	fbExtensionTimeout_TON(IN := bExtending, PT := tExtensionTimeout);	//Timer for monitoring extension timeout, PT = Extension time multiplied by the timeout factor
	fbRetractionTimeout_TON(IN := bRetracting, PT := tRetractionTimeout);	//Timer for monitoring retraction timeout, PT = Retraction time multiplied by the timeout factor

	//Simultaneous extend and retract commands throw an invalid command error
	IF 		(bExtending AND bRetracting)
		OR 	(bExtendRequest AND bRetractRequest)
		OR 	(bExtendCommand AND bRetractCommand) THEN 
		nErrorID := E_CylinderBase.InvalidCommand;
	END_IF
	
	//If both extended and retracted feedback are true at any point, throw an invalid position error
	IF bExtended AND bRetracted THEN
		bError := TRUE;
		nErrorID := E_CylinderBase.InvalidPositionStatus;
	END_IF
	
	//If the cylinder takes longer than expected to extend, throw a timeout error
	IF fbExtensionTimeout_TON.Q THEN
		bError := TRUE;
		nErrorID := E_CylinderBase.ExtendTimeout;
	END_IF
	
	//If the cylinder takes longer than expected to retract, throw a timeout error
	IF fbRetractionTimeout_TON.Q THEN
		bError := TRUE;
		nErrorID := E_CylinderBase.RetractTimeout;
	END_IF
END_IF

//If cylinder is in motion toward a position, but it has not yet been reached, set busy bit
IF (bExtending) OR (bRetracting) THEN
	bActive := TRUE;
ELSE
	bActive := FALSE;
END_IF

IF bSimExtendCommand OR bExtendCommand THEN
	bExtendOutput := TRUE;
ELSE
	bExtendOutput := FALSE;
END_IF

IF bSimRetractCommand OR bRetractCommand THEN
	bRetractOutput := TRUE;
ELSE
	bRetractOutput := FALSE;
END_IF
END_METHOD

METHOD Reset : BOOL
SUPER^.Reset();

bExtending := FALSE;
bRetracting := FALSE;

fbSimExtend_TON.IN := FALSE;
fbSimRetract_TON.IN := FALSE;

bExtendCommand := FALSE;
bRetractCommand := FALSE;
END_METHOD

METHOD Retract : UDINT
bRetractRequest := TRUE;
bExtendRequest := FALSE;
bIncomingRequest := TRUE;
END_METHOD

PROPERTY Retracted : BOOL	//Status bit for the position of the cylinder
GET
Retracted := bRetracted;
END_GET
END_PROPERTY

PROPERTY Retracting : BOOL
GET
Retracting := bRetracting;
END_GET
END_PROPERTY

PROPERTY RetractOutput : BOOL
GET
RetractOutput := bRetractOutput;
END_GET
END_PROPERTY

PROPERTY RetractTime : TIME
GET
RetractTime := tRetractTime;
END_GET
SET
tRetractTime := RetractTime;
END_SET
END_PROPERTY

METHOD SimulateOperation : BOOL
VAR_INPUT
END_VAR
IF bEnabled THEN
	
	bExtendCommand := FALSE;		//Hardware commands should be disabled during simulation mode
	bRetractCommand := FALSE;		//Hardware commands should be disabled during simulation mode
	
	fbSimExtend_TON();		//Call timer FB
	fbSimRetract_TON();		//Call timer FB
	
	IF fbSimExtend_TON.Q THEN		//Whenever the extend timer completes, set status to extended and turn off the timer
		bExtended := TRUE;
		fbSimExtend_TON.IN := FALSE;
	END_IF
	
	IF fbSimRetract_TON.Q THEN		//Whenever the retract timer completes, set status to retracted and turn off the timer
		bRetracted := TRUE;
		fbSimRetract_TON.IN := FALSE;
	END_IF
	
	IF bIncomingRequest THEN
		IF bExtendRequest THEN					//Whenever a new extend request comes in, check to see if we are still currently timing a retract action
			IF fbSimRetract_TON.IN THEN			//If a retract action is still in progress, appropriately scale the extend time to account for the distance traveled during the in-process retraction
				fbSimExtend_TON.PT := tExtendTime * (TIME_TO_UDINT(fbSimRetract_TON.ET) / TIME_TO_UDINT(tRetractTime));		//partial extend time = (full distance extend time) * (proportional distance covered during retraction)
				bSimRetractCommand := FALSE;
				fbSimRetract_TON.IN := FALSE;	//Disable retract timer
			ELSE
				fbSimExtend_TON.PT := tExtendTime;	//If no retraction was active, assume we are currently at fully retracted position, or this is the first command the cylinder has received, so initialize to full extend time
			END_IF
			bRetracted := FALSE;
			bSimRetractCommand := FALSE;
			bSimExtendCommand := TRUE;
			fbSimExtend_TON.IN := TRUE;				//Activate the extension timer
		ELSIF bRetractRequest THEN					//Same as above, but reversed
			IF fbSimExtend_TON.IN THEN
				fbSimRetract_TON.PT := tRetractTime * (TIME_TO_UDINT(fbSimExtend_TON.ET) / TIME_TO_UDINT(tRetractTime));
				bSimExtendCommand := FALSE;
				fbSimExtend_TON.IN := FALSE;
			ELSE
				fbSimRetract_TON.PT := tRetractTime;
			END_IF
			bExtended := FALSE;
			fbSimRetract_TON.IN := TRUE;
			bSimExtendCommand := FALSE;
			bSimRetractCommand := TRUE;
		ELSE
			bExtended := FALSE;
			bRetracted := FALSE;
			
			fbSimExtend_TON.IN := FALSE;			
			fbSimRetract_TON.IN := FALSE;
			
			bSimExtendCommand := FALSE;
			bSimRetractCommand := FALSE;
		END_IF
		bIncomingRequest := FALSE;
	END_IF
	
	bExtending := fbSimExtend_TON.IN;
	bRetracting := fbSimRetract_TON.IN;
ELSE
	bIncomingRequest := FALSE;
	fbSimExtend_TON.IN := FALSE;
	fbSimRetract_TON.IN := FALSE;
END_IF
END_METHOD

METHOD StandardOperation : BOOL
VAR_INPUT
END_VAR
IF bEnabled THEN
	IF bIncomingRequest THEN
		bExtendCommand := bExtendRequest;
		bRetractCommand := bRetractRequest;
		bIncomingRequest := FALSE;
	END_IF
	
	IF bExtendCommand AND NOT bExtended THEN
		bExtending := TRUE;
	END_IF
	
	IF bRetractCommand AND NOT bRetracted THEN
		bRetracting := TRUE;
	END_IF
	
	bExtended := bExtendedFeedback;
	bRetracted := bRetractedFeedback;
ELSE
	bIncomingRequest := FALSE;
END_IF
END_METHOD

PROPERTY TimeoutFactor : LREAL	//Multiplicative factor that determines error timeout threshold based on the expected time
GET
TimeoutFactor := fTimeoutFactor;
END_GET
SET
fTimeoutFactor := TimeoutFactor;
END_SET
END_PROPERTY

END_FUNCTION_BLOCK

// ---- Base/02_Components/01_Base/FB_ComponentBase.TcPOU
FUNCTION_BLOCK FB_ComponentBase IMPLEMENTS ITF_ComponentBase
VAR_INPUT
END_VAR
VAR_OUTPUT
END_VAR
VAR CONSTANT
	//Constant declarations
	COMPONENT_BASE_ALARM_COUNT	: UDINT := 16;
END_VAR

VAR	
	//ITF_BasicComponent internal property variables
	bError 			: BOOL;			//Boolean to signal that an error has ocurred
	nErrorID 		: UDINT;		//Integer ID to identify the proper alarm to be posted from the parent module
	bEnabled		: BOOL;			//Enables or disables the component
	bSimulate		: BOOL;			//TRUE disables all hardware I/O and simulates input and output behavior
	sName			: STRING;		//String name of the component
	bActive			: BOOL;			//TRUE when the component is in its energized state, motion or detection
	
	//Alarming
	a_fbComponentBaseAlarms : ARRAY[1..COMPONENT_BASE_ALARM_COUNT] OF FB_TcAlarm;
	
	//HMI Monitoring and control structure
	stComponentBaseHMI : ST_ComponentBase_HMI;
	
	//Internal Variables
	bInitialized	: BOOL;
	
END_VAR

PROPERTY Active : BOOL	//TRUE when the component is in motion or otherwise completing a commanded task
GET
Active := bActive;
END_GET
END_PROPERTY

METHOD CyclicLogic : BOOL		//Should be called Externally akin to the PML Modules
IF NOT bInitialized THEN
	initialize();
	bInitialized := TRUE;
END_IF

IF NOT bSimulate AND NOT bError THEN	//If not in simulation mode or error state
	StandardOperation();
ELSIF NOT bError THEN
	SimulateOperation();	//Simulate inputs and outputs
ELSE
	ErrorOperation();
END_IF

Monitoring();		//Constant error and status monitoring
HardwareUpdate();	//Passes internal commands to hardware outputs and vice versa for inputs, implement via extended FB override
HMICommunication();	//Keeps the HMI data up to date, and processes requests from the HMI for this component
END_METHOD

PROPERTY Enabled : BOOL	//Enables or disables the component
GET
Enabled := bEnabled;
END_GET
SET
bEnabled := Enabled;
END_SET
END_PROPERTY

PROPERTY Error : BOOL	//Boolean to signal that an error has ocurred
GET
Error := bError;
END_GET
END_PROPERTY

PROPERTY ErrorID : UDINT	//Integer ID to identify the proper alarm to be posted from the parent module
GET
ErrorID := nErrorID;
END_GET
SET
nErrorID := ErrorID;
END_SET
END_PROPERTY

METHOD ErrorOperation : BOOL
VAR_INPUT
END_VAR
//Override from extended FB with error operation logic (Shut off outputs, clear inputs, blink, send error messages, etc)
END_METHOD

METHOD HardwareUpdate : BOOL
VAR_INPUT
END_VAR
//override from extended FB with reads and writes between internal variables and hardware inputs and outputs
END_METHOD

METHOD HMICommunication : BOOL
//Extend this method in extended FBs to communicate specific implementation data

//Process HMI requests
IF stComponentBaseHMI.bIncomingHMIRequest AND NOT stComponentBaseHMI.bHMICommandConfirmation THEN		//If a request has been issued by the HMI, and a previous request has not just finished being processed
	IF stComponentBaseHMI.bHMIControlAvailable THEN		//If the current conditions permit HMI control (Should be determined by the extended application components)
		IF stComponentBaseHMI.bEnableHMIRequest THEN
			bEnabled := TRUE;
			stComponentBaseHMI.bHMICommandConfirmation := TRUE;	//Confirm that the request has been processed
		END_IF
		IF stComponentBaseHMI.bDisableHMIRequest THEN
			bEnabled := FALSE;
			stComponentBaseHMI.bHMICommandConfirmation := TRUE;	//Confirm that the request has been processed
		END_IF
		IF stComponentBaseHMI.bResetHMIRequest THEN
			Reset();
			stComponentBaseHMI.bHMICommandConfirmation := TRUE;	//Confirm that the request has been processed
		END_IF
		IF stComponentBaseHMI.bSimulateOperationHMIRequest THEN
			bSimulate := TRUE;
			stComponentBaseHMI.bHMICommandConfirmation := TRUE;	//Confirm that the request has been processed
		END_IF
		IF stComponentBaseHMI.bStandardOperationHMIRequest THEN
			bSimulate := FALSE;
			stComponentBaseHMI.bHMICommandConfirmation := TRUE;	//Confirm that the request has been processed
		END_IF
	END_IF
END_IF

//Update HMI status info
stComponentBaseHMI.bActive := bActive;
stComponentBaseHMI.bEnabled := bEnabled;
stComponentBaseHMI.sName := sName;
stComponentBaseHMI.bError := bError;
stComponentBaseHMI.bSimulate := bSimulate;
stComponentBaseHMI.nErrorID := nErrorID;
END_METHOD

METHOD initialize : BOOL
VAR_INPUT
END_VAR

VAR
	sTemp: STRING;
END_VAR
//Extend initialize as needed in extended FBs

sTemp := CONCAT(CONCAT(CONCAT('Component ', ': '), sName), ' '); 	//Creates a utility string for alarms and other messaging that reads (example text) - "Module 10 - Main Casepacker" to be followed by the alarm or message info
//TODO: Rename Event Class to AxisBase
F_CreateAllEventsInClass(	p_aAlarms := a_fbComponentBaseAlarms,
							nClassSize := SIZEOF(TC_EVENTS.ComponentBase),
							pInitEvent := ADR(TC_EVENTS.ComponentBase.InitReferenceEvent),
							sPrefix := sTemp );
END_METHOD

METHOD Monitoring : BOOL
VAR_INPUT
END_VAR
//Override/extend from extended FB with monitoring logic
END_METHOD

PROPERTY Name : STRING
GET
Name := sName;
END_GET
SET
sName := Name;
END_SET
END_PROPERTY

METHOD Reset : BOOL
bError := FALSE;
nErrorID := 0;
END_METHOD

{warning 'add property implementation'}
PROPERTY Simulate : BOOL
GET
Simulate := bSimulate;
END_GET
SET
bSimulate := Simulate;
END_SET
END_PROPERTY

METHOD SimulateOperation : BOOL
VAR_INPUT
END_VAR
//Override from extended FB with simulated operation logic
IF bEnabled THEN
	//Do Stuff
	;
ELSE
	//Don't Do Stuff
	;
END_IF
END_METHOD

METHOD StandardOperation : BOOL
VAR_INPUT
END_VAR
//Override from extended FB with normal operation logic
IF bEnabled THEN
	//Do Stuff
	;
ELSE
	//Don't Do Stuff
	;
END_IF
END_METHOD

END_FUNCTION_BLOCK

// ---- Base/02_Components/04_Sensors/02_Sensor/FB_Sensor.TcPOU
FUNCTION_BLOCK FB_Sensor EXTENDS FB_SensorBase
VAR_INPUT
END_VAR
VAR_OUTPUT
END_VAR
VAR
	bSensor_HardwareInput	AT %I* : BOOL;	//Hardware input bit from the hysical sensor
END_VAR

METHOD PRIVATE HardwareUpdate : BOOL
VAR_INPUT
END_VAR
SUPER^.HardwareUpdate();

bRawSensorInput := bSensor_HardwareInput;
END_METHOD

END_FUNCTION_BLOCK

// ---- Base/02_Components/04_Sensors/01_Base/FB_SensorBase.TcPOU
FUNCTION_BLOCK ABSTRACT FB_SensorBase EXTENDS FB_ComponentBase IMPLEMENTS ITF_SensorBase
VAR_INPUT
END_VAR
VAR_OUTPUT
END_VAR
VAR
	//ITF_BasicSensor internal property variables
	eDebounceMode		: E_DebounceMode;	//Defines the debounce model that will filter the sensor's output to the program
	tDebounceTime		: TIME;				//Time input parameter for use in Debounce functionality
	bInverted			: BOOL;				//Defines the output polarity of the sensor - a "TRUE" value will result in the signal of the sensor being inverted
	nSimulationInput	: DINT;				//Provides configuration input to the simulation functionality
	eSimulationMode		: E_SensorSimulationMode;	//Defines the mode of operation for the simulation functionality of this component
	tTimeActive			: TIME;				//Tracks the amount of time that the sensor has been in an active state
	tTimeInactive		: TIME;				//Tracks the amount of time that the sensor has been in an inactive state
	
	//Internal variables
	//bInitialized 			: BOOL;
	fbActiveTimer_TON		: Tc2_Standard.TON;		//Tracks the amount of time that the sensor has been in an active state
	fbInactiveTimer_TON		: Tc2_Standard.TON;		//Tracks the amount of time that the sensor has been in an inactive state
	fbDebounceTimer_TON		: Tc2_Standard.TON;		//Utilized in the debounce implementation
	fbDebounceTimer_TP		: Tc2_Standard.TP;		//Utilized in the debounce implementation
	bRawSensorInput			: BOOL;					//Raw input from sensor
	bProcessedSensorInput	: BOOL;					//Sensor input after Debounce and (if necessary) Inversion
	
	stSensorBaseHMI			: ST_SensorBase_HMI;
	
	//Simulation variables
	bSimulationInput		: DINT;					//Input variable to manipulate simulation behavior
	fbSimulationPulse1_TP	: Tc2_Standard.TP;		//Pulse Timer for simulated sensor pulse generation
	fbSimulationPulse2_TP	: Tc2_Standard.TP;		//Pulse Timer for simulated sensor pulse generation
END_VAR

CyclicLogic();

PROPERTY DebounceMode : E_DebounceMode
GET
DebounceMode := eDebounceMode;
END_GET
SET
eDebounceMode := DebounceMode;
END_SET
END_PROPERTY

PROPERTY DebounceTime : TIME
GET
DebounceTime := tDebounceTime;
END_GET
SET
tDebounceTime := DebounceTime;
END_SET
END_PROPERTY

METHOD HMICommunication : BOOL
SUPER^.HMICommunication();

//Extend this method in extended FBs to communicate specific implementation data

//Process HMI requests
IF stSensorBaseHMI.bIncomingHMIRequest AND NOT stSensorBaseHMI.bHMICommandConfirmation THEN		//If a request has been issued by the HMI, and a previous request has not just finished being processed
	IF stSensorBaseHMI.bHMIControlAvailable THEN		//If the current conditions permit HMI control
		IF stSensorBaseHMI.bSetDebounceModeHMIRequest THEN
			eDebounceMode := stSensorBaseHMI.eSetDebounceModeHMIValue;
			stSensorBaseHMI.bHMICommandConfirmation := TRUE;	//Reset the incoming request bit after the request has been processed
		END_IF
		IF stSensorBaseHMI.bSetDebounceTimeHMIRequest THEN
			tDebounceTime := stSensorBaseHMI.tSetDebounceTimeHMIValue;
			stSensorBaseHMI.bHMICommandConfirmation := TRUE;	//Reset the incoming request bit after the request has been processed
		END_IF
		IF stSensorBaseHMI.bSetSimulationModeHMIRequest THEN
			eSimulationMode := stSensorBaseHMI.eSetSimulationModeHMIValue;
			stSensorBaseHMI.bHMICommandConfirmation := TRUE;	//Reset the incoming request bit after the request has been processed
		END_IF
		IF stSensorBaseHMI.bSetSimulationInputHMIRequest THEN
			nSimulationInput := stSensorBaseHMI.nSetSimulationInputHMIValue;
			stSensorBaseHMI.bHMICommandConfirmation := TRUE;	//Reset the incoming request bit after the request has been processed
		END_IF
		IF stSensorBaseHMI.bInvertedHMIRequest THEN
			bInverted := TRUE;
			stSensorBaseHMI.bHMICommandConfirmation := TRUE;	//Reset the incoming request bit after the request has been processed
		END_IF
		IF stSensorBaseHMI.bUninvertedHMIRequest THEN
			bInverted := FALSE;
			stSensorBaseHMI.bHMICommandConfirmation := TRUE;	//Reset the incoming request bit after the request has been processed
		END_IF
		IF stSensorBaseHMI.bSimulateOperationHMIRequest THEN
			bSimulate := TRUE;
			stSensorBaseHMI.bHMICommandConfirmation := TRUE;	//Reset the incoming request bit after the request has been processed
		END_IF
		IF stSensorBaseHMI.bStandardOperationHMIRequest THEN
			bSimulate := FALSE;
			stSensorBaseHMI.bHMICommandConfirmation := TRUE;	//Reset the incoming request bit after the request has been processed
		END_IF
	END_IF
END_IF

//Update HMI status info
stSensorBaseHMI.eDebounceMode := eDebounceMode;
stSensorBaseHMI.tDebounceTime := tDebounceTime;
stSensorBaseHMI.bInverted := bInverted;
stSensorBaseHMI.eSimulationMode := eSimulationMode;
stSensorBaseHMI.nSimulationInput := nSimulationInput;
stSensorBaseHMI.tTimeActive := tTimeActive;
stSensorBaseHMI.tTimeInactive := tTimeInactive;
END_METHOD

METHOD InitialConfig : BOOL
VAR_INPUT	
	eDBMode				: E_DebounceMode;			//Debounce Mode
	tDBTime				: TIME;						//Debounce Time
	bEnable			: BOOL;						//Enable or Disable the sensor's operation
	bInvert			: BOOL;						//TRUE = Invert return signal
	bSim			: BOOL;						//TRUE = Ignore Hardware and simulate sensor operation
	nSimInput 	: DINT;						//Input parameter for simulation adjustment
	eSimMode		: E_SensorSimulationMode;	//Configure Simulation behavior of the sensor
END_VAR
DebounceMode := eDBMode;
DebounceTime := tDBTime;
Enabled := bEnable;
Inverted := bInvert;
Simulate := bSim;
SimulationInput := nSimInput;
SimulationMode := eSimMode;
END_METHOD

PROPERTY Inverted : BOOL
GET
Inverted := bInverted;
END_GET
SET
bInverted := Inverted;
END_SET
END_PROPERTY

METHOD Monitoring : BOOL
VAR_INPUT
END_VAR
SUPER^.Monitoring();

//If flicker counters or other diagnostic systems are desired, their implementation could be here
//Any warnings, errors, or other desired messages would also be generated here

//T#71582M47S295MS is the upper bound of the TIME type, meaning these timers will continue to increase ET for as long as possible
fbActiveTimer_TON(IN := bActive, PT := T#71582M47S295MS, ET => tTimeActive);
fbInactiveTimer_TON(IN := NOT bActive, PT := T#71582M47S295MS, ET => tTimeInactive);
END_METHOD

METHOD ProcessInput : BOOL
VAR_INPUT
	bInput	: BOOL;
END_VAR
VAR
	bDebouncedInput	: BOOL;
END_VAR
VAR_INST
	bLastDebouncedInput : BOOL;
	nMovingAverage		: DINT;
END_VAR
CASE eDebounceMode OF
	E_DebounceMode.RawInput:					//Passes raw input through
		bDebouncedInput := bInput;		
		
	E_DebounceMode.SimpleFlickerFilter:			//Requires the raw input to be a consistent value for a set time period before output changes
		fbDebounceTimer_TON(IN := (bInput <> bDebouncedInput), PT := tDebounceTime);	//runs the timer whenever a differing input is detected
		IF fbDebounceTimer_TON.Q THEN
			bDebouncedInput := bInput;	//once the raw input has been different for the specified debounce time, the processed input is updated
		END_IF
	E_DebounceMode.EdgeDetectFilter:			//Updates the processed value immediately on a change from steady state, but mutes any sensor flickers for the specified time immediately following the change
		IF (bInput <> bDebouncedInput) AND (NOT fbDebounceTimer_TP.Q) THEN			//A differing raw input must be detected outside of the mute window created by the pulse timer
			bDebouncedInput := bInput;
		END_IF
		fbDebounceTimer_TP(IN := (bDebouncedInput <> bLastDebouncedInput), PT := tDebounceTime);	//"Q" will be TRUE for tDebounce time after the bProcessedSensorInput value is changed
	E_DebounceMode.MovingAverage:		//Uses a "moving average"-like calculation to compensate for extremely inconsistent signals - prevents poorly timed flickers from causing disproportionate results
		fbDebounceTimer_TON(IN := NOT fbDebounceTimer_TON.Q, PT := T#5MS);	//Provides a 1ms "polling" trigger
		IF fbDebounceTimer_TON.Q THEN		//TRUE once every millisecond
			IF bInput THEN			//If raw input is currently active at the time of polling
				IF nMovingAverage < TIME_TO_DINT(tDebounceTime) THEN	//If the moving average has not reached its "weight limit" as set by debounce time
					nMovingAverage := nMovingAverage + 5;		//Add 1 to the average
				END_IF
			ELSE	//If raw input is currently inactive at the time of polling
				IF nMovingAverage > - TIME_TO_DINT(tDebounceTime) THEN	//If the moving average has not reached its "weight limit" as set by debounce time
					nMovingAverage := nMovingAverage - 5;		//Subtract 1 from the average
				END_IF
			END_IF
		END_IF
		
		IF nMovingAverage >= 0 THEN
			bDebouncedInput := TRUE;
		ELSE
			bDebouncedInput := FALSE;
		
		END_IF
END_CASE

bLastDebouncedInput := bDebouncedInput;		//Update "Last value"

IF bInverted THEN		//If signal inversion is requested, invert the signal
	bProcessedSensorInput := NOT bDebouncedInput;
ELSE 
	bProcessedSensorInput := bDebouncedInput;
END_IF
END_METHOD

METHOD SimulateOperation : BOOL
VAR_INPUT
END_VAR
CASE eSimulationMode OF
	E_SensorSimulationMode.InputDriven:
		ProcessInput(bInput := DINT_TO_BOOL(bSimulationInput));
	E_SensorSimulationMode.Periodic:
		fbSimulationPulse1_TP(IN := NOT fbSimulationPulse2_TP.Q, PT := DINT_TO_TIME(nSimulationInput));
		fbSimulationPulse2_TP(IN := NOT fbSimulationPulse1_TP.Q, PT := DINT_TO_TIME(nSimulationInput));
		ProcessInput(bInput := fbSimulationPulse2_TP.Q);
END_CASE

bActive := bProcessedSensorInput;
END_METHOD

PROPERTY SimulationInput : DINT
GET
SimulationInput := nSimulationInput;
END_GET
SET
nSimulationInput := SimulationInput;
END_SET
END_PROPERTY

PROPERTY SimulationMode : E_SensorSimulationMode
GET
SimulationMode := eSimulationMode;
END_GET
SET
eSimulationMode := SimulationMode;
END_SET
END_PROPERTY

METHOD StandardOperation : BOOL
VAR_INPUT
END_VAR
ProcessInput(bInput := bRawSensorInput);
bActive := bProcessedSensorInput;
END_METHOD

PROPERTY TimeActive : TIME
GET
TimeActive := tTimeActive;
END_GET
END_PROPERTY

PROPERTY TimeInactive : TIME
GET
TimeInactive := tTimeInactive;
END_GET
END_PROPERTY

END_FUNCTION_BLOCK

// ---- Base/02_Components/02_Axes/03_MotionType/FB_Axis_Continuous_NoHoming.TcPOU
FUNCTION_BLOCK FB_Axis_Continuous_NoHoming EXTENDS FB_Axis_NoHoming IMPLEMENTS ITF_Axis_Continuous
VAR_INPUT
END_VAR
VAR_OUTPUT
END_VAR
VAR
	//Internal Property Variables
	fModuloPosition		: LREAL;
	fModuloFactor		: LREAL;
END_VAR

PROPERTY ModuloFactor : LREAL
GET
ModuloFactor := fModuloFactor;
END_GET
END_PROPERTY

PROPERTY ModuloPosition : LREAL
GET
ModuloPosition := fModuloPosition;
END_GET
END_PROPERTY

METHOD Monitoring : BOOL
SUPER^.Monitoring();

fModuloPosition := SelectedAxis.NcToPlc.ModuloActPos;

IF fbWriteParameter.Done AND fbWriteParameter.ParameterNumber = MC_AxisParameter.AxisEncoderModuloValue THEN
	fModuloFactor := fbWriteParameter.Value;
END_IF

IF fbWriteParameter.Error AND NOT fbAxisBaseAlarms[E_AxisBase.WriteParameterError].bRaised THEN
	bError := TRUE;
	nErrorID := E_AxisBase.WriteParameterError;
	sTemp := UDINT_TO_STRING(fbWriteParameter.ErrorID);
	fbAxisBaseAlarms[E_AxisBase.WriteParameterError].ipArguments.Clear().AddString(sName).AddString(sTemp);
	fbAxisBaseAlarms[E_AxisBase.WriteParameterError].Raise(0);
ELSIF NOT fbAxisPower.Error AND fbAxisBaseAlarms[E_AxisBase.WriteParameterError].bRaised THEN
	fbAxisBaseAlarms[E_AxisBase.WriteParameterError].Clear(0,0);
END_IF
END_METHOD

METHOD SetAxisModuloFactor : BOOL
VAR_INPUT
	fSetAxisModuloFactor		: LREAL;
END_VAR
IF NOT bActive THEN
	IF NOT fbWriteParameter.Busy THEN
	fbWriteParameter(
						Axis:= SelectedAxis, 
						Execute:= TRUE, 
						ParameterNumber:= MC_AxisParameter.AxisEncoderModuloValue, 
						Value:= fSetAxisModuloFactor, 
						Done=> , 
						Busy=> , 
						Error=> , 
						ErrorID=> );
	END_IF
ELSE
	//TODO: Messaging for "Axis not ready for parameter write"
END_IF
END_METHOD

END_FUNCTION_BLOCK

// ---- Base/02_Components/02_Axes/02_Homing/FB_Axis_NoHoming.TcPOU
FUNCTION_BLOCK FB_Axis_NoHoming EXTENDS FB_AxisBase
VAR_INPUT
END_VAR
VAR_OUTPUT
END_VAR
VAR
END_VAR

METHOD MotionControl : BOOL
VAR_INPUT
END_VAR
SUPER^.MotionControl();

IF bDriveEnabled AND NOT SelectedAxis.Status.Homed THEN
	//Since homing does not matter for this axis, just home it wherever it sits when enabled
	fbAxisHome(
				Axis:= SelectedAxis, 
				Execute:= TRUE, 
				Position:= 0, 
				HomingMode:= MC_Direct, 
				BufferMode:= , 
				Options:= , 
				bCalibrationCam:= TRUE, 
				Done=> , 
				Busy=> , 
				Active=> , 
				CommandAborted=> , 
				Error=> , 
				ErrorID=> );
END_IF
END_METHOD

END_FUNCTION_BLOCK

// ---- Base/02_Components/02_Axes/01_Base/FB_AxisBase.TcPOU
FUNCTION_BLOCK ABSTRACT FB_AxisBase EXTENDS FB_ComponentBase IMPLEMENTS ITF_AxisBase
VAR CONSTANT
	//Constant declarations
	AXIS_BASE_ALARM_COUNT	: UDINT := 16;
END_VAR

VAR
	//ITF_AxisBase internal property variables
	fJogFastVelocity	: LREAL;
	fJogSlowVelocity	: LREAL;
	fTargetVelocity		: LREAL;
	
	bDriveEnabled		: BOOL;
	bInGear				: BOOL;
	bInPosition			: BOOL;
	fPosition 			: LREAL;
	fPositionSetpoint	: LREAL;
	bStopped			: BOOL;
	
	//Axis MC function blocks
	fbAxisJog: MC_Jog;
	fbAxisPower: MC_Power;
	fbAxisReset: MC_Reset;
	fbMoveAbsolute: MC_MoveAbsolute;
	fbMoveVelocity: MC_MoveVelocity;
	fbMoveRelative: MC_MoveRelative;
	fbAxisHalt: MC_Halt;
	fbAxisStop: MC_Stop;
	fbAxisHome: MC_Home;
	fbGearIn: MC_GearIn;
	fbResetDrv: FB_SoEReset;
	fbWriteParameter : MC_WriteParameter;
	
	//Alarming
	fbAxisBaseAlarms : ARRAY[1..AXIS_BASE_ALARM_COUNT] OF FB_TcAlarm;
	
	//Internal Variables
	fOverride		: LREAL := 100;		//Velocity Override
	SelectedAxis	: REFERENCE TO AXIS_REF REF= SimulationAxis;	//TODO: Make a better simulation system
	SimulationAxis: AXIS_REF;
	HardwareAxis: AXIS_REF;

	sTemp: STRING;
	stAxisBaseHMI		: ST_AxisBase_HMI;
	
	nAxisCopy: INT;
	bParamCopyComplete: BOOL;
END_VAR
VAR_IN_OUT
	MasterAxis	: AXIS_REF;
END_VAR

PROPERTY AxisRef : AXIS_REF
GET
AxisRef := SelectedAxis;
END_GET
END_PROPERTY

PROPERTY DriveEnabled : BOOL
GET
Enabled := bDriveEnabled;
END_GET
END_PROPERTY

METHOD ErrorOperation : BOOL
VAR_INPUT
END_VAR
SUPER^.ErrorOperation();

bEnabled := FALSE;
END_METHOD

METHOD GearInBasic : BOOL
VAR_IN_OUT
	master : AXIS_REF;	//Master axis to which the gearing will be made
END_VAR
IF NOT bActive THEN
	
	MasterAxis := master;		//"Master" must be specified in the FB call, so this particular variable is declared in the main FB and assigned from here
	fbGearIn.Execute := TRUE;
	
END_IF
END_METHOD

METHOD HardwareUpdate : BOOL
VAR_INPUT
END_VAR
SUPER^.HardwareUpdate();
	
//Resets the axis Drive Hardware when commanded by a "ResetDrive" Method call
fbResetDrv(
	NetId:= '', 
	Timeout:= T#10S, 
	Axis:= HardwareAxis);
	
fbResetDrv.Execute := FALSE;
END_METHOD

METHOD HMICommunication : BOOL
//Extend this method in extended FBs to communicate specific implementation data
SUPER^.HMICommunication();

//Process HMI requests
IF stAxisBaseHMI.bIncomingHMIRequest AND NOT stAxisBaseHMI.bHMICommandConfirmation THEN		//If a request has been issued by the HMI, and a previous request has not just finished being processed
	IF stAxisBaseHMI.bHMIControlAvailable THEN		//If the current conditions permit HMI control (Should be determined by the extended application components)
		IF stAxisBaseHMI.bDriveEnableHMIRequest THEN
			bEnabled := TRUE;
			stAxisBaseHMI.bHMICommandConfirmation := TRUE;	//Confirm that the request has been processed
		END_IF
		IF stAxisBaseHMI.bDriveDisableHMIRequest THEN
			bEnabled := FALSE;
			stAxisBaseHMI.bHMICommandConfirmation := TRUE;	//Confirm that the request has been processed
		END_IF
		IF stAxisBaseHMI.bSetJogFastVelocityRequest THEN
			fJogFastVelocity := stAxisBaseHMI.fSetJogFastVelocityValue;
			stAxisBaseHMI.bHMICommandConfirmation := TRUE;	//Confirm that the request has been processed
		END_IF
		IF stAxisBaseHMI.bSetJogSlowVelocityRequest THEN
			fJogSlowVelocity := stAxisBaseHMI.fSetJogSlowVelocityValue;
			stAxisBaseHMI.bHMICommandConfirmation := TRUE;	//Confirm that the request has been processed
		END_IF
		IF stAxisBaseHMI.bSetTargetVelocityRequest THEN
			fTargetVelocity := stAxisBaseHMI.bSetTargetVelocityValue;
			stAxisBaseHMI.bHMICommandConfirmation := TRUE;	//Confirm that the request has been processed
		END_IF
	END_IF
END_IF

//Update HMI status info
stAxisBaseHMI.fJogFastVelocity := fJogFastVelocity;
stAxisBaseHMI.fJogSlowVelocity := fJogSlowVelocity;
stAxisBaseHMI.fTargetVelocity := fTargetVelocity;
stAxisBaseHMI.bDriveEnabled := bDriveEnabled;
stAxisBaseHMI.bInGear := bInGear;
stAxisBaseHMI.bInPosition := bInPosition;
stAxisBaseHMI.fPosition := fPosition;
stAxisBaseHMI.fPositionSetpoint := fPositionSetpoint;
stAxisBaseHMI.bStopped := bStopped;
END_METHOD

METHOD Home : BOOL
//This method should be overridden by the extending FB based on the specific hardware configuration
END_METHOD

PROPERTY InGear : BOOL
GET
InGear := bInGear;
END_GET
END_PROPERTY

METHOD Inhibit : BOOL
VAR_INPUT
END_VAR
fbAxisPower.Override := 0;
END_METHOD

METHOD initialize : BOOL
VAR_INPUT
END_VAR

VAR
	sTemp: STRING;
END_VAR
SUPER^.initialize();

sTemp := CONCAT(CONCAT(CONCAT('Axis ', ': '), sName), ' '); 	//Creates a utility string for alarms and other messaging that reads (example text) - "Module 10 - Main Casepacker" to be followed by the alarm or message info
//TODO: Rename Event Class to AxisBase
F_CreateAllEventsInClass(	p_aAlarms := fbAxisBaseAlarms,
							nClassSize := SIZEOF(TC_EVENTS.AxisBase),
							pInitEvent := ADR(TC_EVENTS.AxisBase.InitReferenceEvent),
							sPrefix := sTemp );
END_METHOD

PROPERTY InPosition : BOOL
GET
InPosition := bInPosition;
END_GET
END_PROPERTY

METHOD Jog : BOOL
VAR_INPUT
	direction	: BOOL;			//"TRUE" for positive jog, "FALSE" for negative jog
	fast		: BOOL;			//"TRUE" for 'fast' jog, "FALSE" for 'slow' jog (As defined by Jog(Slow/Fast)Velocity Property)
END_VAR
//If the jog is currently active, allow the method to run again to ensure that the corresponding Jog bit can remain high so the jog can continue
//Otherwise, only start a jog when the axis is not already busy
IF fbAxisJog.Busy OR NOT bActive THEN
	
	fbAxisJog.JogForward:= direction; 
	fbAxisJog.JogBackwards:= NOT direction;
	
	IF fast THEN
		fbAxisJog.Velocity := fJogFastVelocity;
	ELSE
		fbAxisJog.Velocity := fJogSlowVelocity;
	END_IF
	
END_IF
END_METHOD

PROPERTY JogFastVelocity : LREAL
GET
JogFastVelocity : fJogFastVelocity;
END_GET
SET
fJogFastVelocity := JogFastVelocity;
END_SET
END_PROPERTY

PROPERTY JogSlowVelocity : LREAL
GET
JogSlowVelocity : fJogSlowVelocity;
END_GET
SET
fJogSlowVelocity : JogSlowVelocity;
END_SET
END_PROPERTY

METHOD Monitoring : BOOL
SUPER^.Monitoring();

//Cyclically updates the "Status" values from the NC-axis to the PLC (Axis1.Status...)
SelectedAxis.ReadStatus();

//Cyclically monitor all FB "Busy" bits, as well as the axis "HasJob" bit to ensure ADS communication time does not result in a delay before the "Busy" property is accurate after calling a FB
bActive := 		SimulationAxis.Status.HasJob
				OR	fbAxisJog.Busy
				OR	fbMoveAbsolute.Busy
				OR	fbMoveVelocity.Busy
				OR	fbMoveRelative.Busy
				OR	fbAxisHalt.Busy
				OR	fbAxisStop.Busy
				OR	fbAxisHome.Busy
				OR	fbGearIn.Busy;
				

//Update all internal property variables
bDriveEnabled := fbAxisPower.Status;
bInGear	:= (SelectedAxis.NcToPlc.CoupleState = 3);	//Note that this only looks for a simple gearing arrangement where this axis is a slave and not a master to any other axis
bInPosition := SelectedAxis.Status.InTargetPosition;
fPosition := SelectedAxis.NcToPlc.ActPos;
fPositionSetpoint := SelectedAxis.NcToPlc.SetPos;
bStopped := SelectedAxis.Status.StandStill;

				
//Error monitoring and event logging

IF fbAxisJog.Error AND NOT fbAxisBaseAlarms[E_AxisBase.JogError].bRaised THEN
	bError := TRUE;
	nErrorID := E_AxisBase.JogError;
	sTemp := UDINT_TO_STRING(fbAxisJog.ErrorID);
	fbAxisBaseAlarms[E_AxisBase.JogError].ipArguments.Clear().AddString(sName).AddString(sTemp);
	fbAxisBaseAlarms[E_AxisBase.JogError].Raise(0);
ELSIF NOT fbAxisJog.Error AND fbAxisBaseAlarms[E_AxisBase.JogError].bRaised THEN
	fbAxisBaseAlarms[E_AxisBase.JogError].Clear(0,0);
END_IF


IF fbAxisPower.Error AND NOT fbAxisBaseAlarms[E_AxisBase.PowerError].bRaised THEN
	bError := TRUE;
	nErrorID := E_AxisBase.PowerError;
	sTemp := UDINT_TO_STRING(fbAxisPower.ErrorID);
	fbAxisBaseAlarms[E_AxisBase.PowerError].ipArguments.Clear().AddString(sName).AddString(sTemp);
	fbAxisBaseAlarms[E_AxisBase.PowerError].Raise(0);
ELSIF NOT fbAxisPower.Error AND fbAxisBaseAlarms[E_AxisBase.PowerError].bRaised THEN
	fbAxisBaseAlarms[E_AxisBase.PowerError].Clear(0,0);
END_IF


IF fbAxisReset.Error AND NOT fbAxisBaseAlarms[E_AxisBase.ResetError].bRaised THEN
	bError := TRUE;
	nErrorID := E_AxisBase.ResetError;
	sTemp := UDINT_TO_STRING(fbAxisReset.ErrorID);
	fbAxisBaseAlarms[E_AxisBase.ResetError].ipArguments.Clear().AddString(sName).AddString(sTemp);
	fbAxisBaseAlarms[E_AxisBase.ResetError].Raise(0);
ELSIF NOT fbAxisReset.Error AND fbAxisBaseAlarms[E_AxisBase.ResetError].bRaised THEN
	fbAxisBaseAlarms[E_AxisBase.ResetError].Clear(0,0);
END_IF


IF fbMoveAbsolute.Error AND NOT fbAxisBaseAlarms[E_AxisBase.MoveAbsoluteError].bRaised THEN
	bError := TRUE;
	nErrorID := E_AxisBase.MoveAbsoluteError;
	sTemp := UDINT_TO_STRING(fbMoveAbsolute.ErrorID);
	fbAxisBaseAlarms[E_AxisBase.MoveAbsoluteError].ipArguments.Clear().AddString(sName).AddString(sTemp);
	fbAxisBaseAlarms[E_AxisBase.MoveAbsoluteError].Raise(0);
ELSIF NOT fbMoveAbsolute.Error AND fbAxisBaseAlarms[E_AxisBase.MoveAbsoluteError].bRaised THEN
	fbAxisBaseAlarms[E_AxisBase.MoveAbsoluteError].Clear(0,0);
END_IF


IF fbMoveVelocity.Error AND NOT fbAxisBaseAlarms[E_AxisBase.MoveVelocityError].bRaised THEN
	bError := TRUE;
	nErrorID := E_AxisBase.MoveVelocityError;
	sTemp := UDINT_TO_STRING(fbMoveVelocity.ErrorID);
	fbAxisBaseAlarms[E_AxisBase.MoveVelocityError].ipArguments.Clear().AddString(sName).AddString(sTemp);
	fbAxisBaseAlarms[E_AxisBase.MoveVelocityError].Raise(0);
ELSIF NOT fbMoveVelocity.Error AND fbAxisBaseAlarms[E_AxisBase.MoveVelocityError].bRaised THEN
	fbAxisBaseAlarms[E_AxisBase.MoveVelocityError].Clear(0,0);
END_IF


IF fbMoveRelative.Error AND NOT fbAxisBaseAlarms[E_AxisBase.MoveRelativeError].bRaised THEN
	bError := TRUE;
	nErrorID := E_AxisBase.MoveRelativeError;
	sTemp := UDINT_TO_STRING(fbMoveRelative.ErrorID);
	fbAxisBaseAlarms[E_AxisBase.MoveRelativeError].ipArguments.Clear().AddString(sName).AddString(sTemp);
	fbAxisBaseAlarms[E_AxisBase.MoveRelativeError].Raise(0);
ELSIF NOT fbMoveRelative.Error AND fbAxisBaseAlarms[E_AxisBase.MoveRelativeError].bRaised THEN
	fbAxisBaseAlarms[E_AxisBase.MoveRelativeError].Clear(0,0);
END_IF


IF fbAxisHalt.Error AND NOT fbAxisBaseAlarms[E_AxisBase.HaltError].bRaised THEN
	bError := TRUE;
	nErrorID := E_AxisBase.HaltError;
	sTemp := UDINT_TO_STRING(fbAxisHalt.ErrorID);
	fbAxisBaseAlarms[E_AxisBase.HaltError].ipArguments.Clear().AddString(sName).AddString(sTemp);
	fbAxisBaseAlarms[E_AxisBase.HaltError].Raise(0);
ELSIF NOT fbAxisHalt.Error AND fbAxisBaseAlarms[E_AxisBase.HaltError].bRaised THEN
	fbAxisBaseAlarms[E_AxisBase.HaltError].Clear(0,0);
END_IF


IF fbAxisStop.Error AND NOT fbAxisBaseAlarms[E_AxisBase.StopError].bRaised THEN
	bError := TRUE;
	nErrorID := E_AxisBase.StopError;
	sTemp := UDINT_TO_STRING(fbAxisStop.ErrorID);
	fbAxisBaseAlarms[E_AxisBase.StopError].ipArguments.Clear().AddString(sName).AddString(sTemp);
	fbAxisBaseAlarms[E_AxisBase.StopError].Raise(0);
ELSIF NOT fbAxisStop.Error AND fbAxisBaseAlarms[E_AxisBase.StopError].bRaised THEN
	fbAxisBaseAlarms[E_AxisBase.StopError].Clear(0,0);
END_IF


IF fbAxisHome.Error AND NOT fbAxisBaseAlarms[E_AxisBase.HomeError].bRaised THEN
	bError := TRUE;
	nErrorID := E_AxisBase.HomeError;
	sTemp := UDINT_TO_STRING(fbAxisHome.ErrorID);
	fbAxisBaseAlarms[E_AxisBase.HomeError].ipArguments.Clear().AddString(sName).AddString(sTemp);
	fbAxisBaseAlarms[E_AxisBase.HomeError].Raise(0);
ELSIF NOT fbAxisHome.Error AND fbAxisBaseAlarms[E_AxisBase.HomeError].bRaised THEN
	fbAxisBaseAlarms[E_AxisBase.HomeError].Clear(0,0);
END_IF


IF fbGearIn.Error AND NOT fbAxisBaseAlarms[E_AxisBase.GearInError].bRaised THEN
	bError := TRUE;
	nErrorID := E_AxisBase.GearInError;
	sTemp := UDINT_TO_STRING(fbGearIn.ErrorID);
	fbAxisBaseAlarms[E_AxisBase.GearInError].ipArguments.Clear().AddString(sName).AddString(sTemp);
	fbAxisBaseAlarms[E_AxisBase.GearInError].Raise(0);
ELSIF NOT fbGearIn.Error AND fbAxisBaseAlarms[E_AxisBase.GearInError].bRaised THEN
	fbAxisBaseAlarms[E_AxisBase.GearInError].Clear(0,0);
END_IF


IF fbResetDrv.Error AND NOT fbAxisBaseAlarms[E_AxisBase.ResetError].bRaised THEN
	bError := TRUE;
	nErrorID := E_AxisBase.ResetError;
	sTemp := UDINT_TO_STRING(fbResetDrv.AdsErrId);
	fbAxisBaseAlarms[E_AxisBase.ResetError].ipArguments.Clear().AddString(sName).AddString(sTemp);
	fbAxisBaseAlarms[E_AxisBase.ResetError].Raise(0);
ELSIF NOT fbResetDrv.Error AND fbAxisBaseAlarms[E_AxisBase.ResetError].bRaised THEN
	fbAxisBaseAlarms[E_AxisBase.ResetError].Clear(0,0);
END_IF

IF fbAxisPower.Override = 0 AND bActive AND NOT fbAxisBaseAlarms[E_AxisBase.CommandWhileInhibited].bRaised THEN
	bError := TRUE;
	nErrorID := E_AxisBase.CommandWhileInhibited;
	fbAxisBaseAlarms[E_AxisBase.CommandWhileInhibited].Raise(0);
ELSIF fbAxisPower.Override <> 0 AND fbAxisBaseAlarms[E_AxisBase.CommandWhileInhibited].bRaised THEN
	fbAxisBaseAlarms[E_AxisBase.CommandWhileInhibited].Clear(0,0);
END_IF

IF SimulationAxis.Status.Error AND NOT fbAxisBaseAlarms[E_AxisBase.DriveError].bRaised THEN
	bError := TRUE;
	nErrorID := E_AxisBase.DriveError;
	sTemp := UDINT_TO_STRING(SimulationAxis.Status.ErrorID);
	fbAxisBaseAlarms[E_AxisBase.DriveError].ipArguments.Clear().AddString(sName).AddString(sTemp);
	fbAxisBaseAlarms[E_AxisBase.DriveError].Raise(0);
END_IF
END_METHOD

METHOD MotionControl : BOOL
VAR_INPUT
END_VAR
//Enables the Axis for movement when commanded by an "Enable" Method call
fbAxisPower(
	Axis:= SelectedAxis,
	Enable:= bEnabled AND (bParamCopyComplete OR NOT bSimulate),
	Enable_Positive:= TRUE, 
	Enable_Negative:= TRUE, 
	Override:= fOverride, 
	BufferMode:= MC_BufferMode.MC_Aborting);


//Cyclically calls all motion fbs so that they can properly communicate to the NC
//Trigger bits (usually "Execute") are set false after each block so that external setting of execute will be read and then cleared without requiring external monitoring

//Moves the Axis to a Set Position when commanded by a "MovePosition" Method call
fbMoveAbsolute(
	Axis:= SelectedAxis,
	Velocity:= fTargetVelocity, 
	BufferMode:= MC_BufferMode.MC_Aborting );
	
fbMoveAbsolute.Execute := FALSE;

//Moves the Axis a Set Distance from its current position when commanded by a "MoveRelative" Method call
fbMoveRelative(
	Axis:= SelectedAxis, 
	Velocity:= fTargetVelocity, 
	BufferMode:= MC_BufferMode.MC_Aborting );

fbMoveRelative.Execute := FALSE;

//Starts a continuous move at a set velocity when commanded by a "MoveVelocity" Method call
fbMoveVelocity(
	Axis:= SelectedAxis, 
	Direction:= MC_Direction.MC_Positive_Direction, 
	BufferMode:= MC_BufferMode.MC_Aborting );	

fbMoveVelocity.Execute := FALSE;

//Performs a simple "Gearing" of the axis to a specified master axis at 1:1 ratio
fbGearIn(
	Master:= MasterAxis, 
	Slave:= SelectedAxis, 
	RatioNumerator:= 1, 
	RatioDenominator:= 1);
	
fbGearIn.Execute := FALSE;

//Halts the axis without disabling future commands when commanded by the "Stop" Method call
fbAxisHalt(
	Axis:= SelectedAxis,  
	BufferMode:= MC_BufferMode.MC_Aborting );	
	
fbAxisHalt.Execute := FALSE;

//Jogs the axis in a specified direction and velocity when commanded by a "Jog" Method call
fbAxisJog(
	Axis:= SelectedAxis,  
	Mode:= E_JogMode.MC_JOGMODE_CONTINOUS);

fbAxisJog.JogForward := FALSE;		//While the Jog FB does require a constant input in Continuous mode, the Method code will happen between here and the fb being called again, so the FB will not see this blip to false
fbAxisJog.JogBackwards := FALSE;	//When the "Jog" method is no longer being called, this will ensure that the jog stops on the next program cycle

//Resets the NC software axis when commanded by a "Reset" Method call
fbAxisReset(
	Axis:= SelectedAxis);

fbAxisReset.Execute := FALSE;
END_METHOD

METHOD MovePosition : BOOL
VAR_INPUT
	override 	: BOOL := FALSE;		//Allows this instruction to override another ongoing operation(This parameter is initialized so that once default parameter value functionality is added to TwinCAT, this input will not need to be set explicitly in the Method call)
	position	: LREAL;				//Desired position to which the axis should move
END_VAR
IF override OR NOT bActive THEN
	
	fbMoveAbsolute.Position := position;
	fbMoveAbsolute.Execute := TRUE;
	
END_IF
END_METHOD

METHOD MoveRelative : BOOL
VAR_INPUT
	override 	: BOOL := FALSE;		//Allows this instruction to override another ongoing operation(This parameter is initialized so that once default parameter value functionality is added to TwinCAT, this input will not need to be set explicitly in the Method call)
	distance 	: LREAL;				//Desired distance to be moved
END_VAR
IF override OR NOT bActive THEN
	
	fbMoveRelative.Distance := distance;
	fbMoveRelative.Execute := TRUE;
	
END_IF
END_METHOD

METHOD MoveVelocity : BOOL
VAR_INPUT
	override	: BOOL := FALSE;				//Allows this instruction to override another ongoing operation(This parameter is initialized so that once default parameter value functionality is added to TwinCAT, this input will not need to be set explicitly in the Method call)
	velocity	: LREAL := fTargetVelocity;		//Desired velocity for the axis (This parameter is initialized so that once default parameter value functionality is added to TwinCAT, this input will not need to be set explicitly in the Method call)
END_VAR
IF override OR NOT bActive THEN
	
	fbMoveVelocity.Velocity := velocity;
	fbMoveVelocity.Execute := TRUE;
	
END_IF
END_METHOD

PROPERTY Position : LREAL
GET
Position := fPosition;
END_GET
END_PROPERTY

PROPERTY PositionSetpoint : LREAL
GET
PositionSetpoint := fPositionSetpoint;
END_GET
END_PROPERTY

METHOD Reset : BOOL
SUPER^.Reset();

fbAxisReset.Execute := TRUE;
fbResetDrv.Execute := TRUE;
END_METHOD

METHOD ResetDrive : BOOL
fbResetDrv.Execute := FALSE;
END_METHOD

PROPERTY Simulate : BOOL
GET
END_GET
SET
END_SET
END_PROPERTY

METHOD SimulateOperation : BOOL
VAR_INPUT
END_VAR
VAR_INST
	fbWriteParam: ARRAY[1..8] OF MC_WriteParameter;
	fbAxisParamRead : ARRAY[1..8] OF MC_ReadParameter;
	fTestValue: LREAL;
	fbSetSimulationPosition: MC_SetPosition;
END_VAR
VAR
	i: INT;
END_VAR
// the need is to insure that the simulation axis always has the same dynamics and speed setpoints as the hardware axis
//copy sequence using MC2 Function Blocks

CASE nAxisCopy OF
	0:	// hold state waiting to start
		FOR i := 1 TO 8 DO
			fbAxisParamRead[i](
				Axis:= HardwareAxis,
				Enable := FALSE);
			fbWriteParam[i](
				Axis:=SimulationAxis , 
				Execute:= FALSE);
		END_FOR
		
		nAxisCopy := 10;
	10:	//read axis param
		bParamCopyComplete := FALSE;
		fbAxisParamRead[1](
			Axis:= HardwareAxis, 
			Enable:=TRUE , 
			ParameterNumber:= MC_AxisParameter.AxisMaxVelocity, 
			ReadMode:= 1, 
				Value=> fTestValue );
		fbAxisParamRead[2](
			Axis:= HardwareAxis, 
			Enable:=TRUE , 
			ParameterNumber:= MC_AxisParameter.AxisAcc, 
			ReadMode:= 1 );
		fbAxisParamRead[3](
			Axis:= HardwareAxis, 
			Enable:=TRUE , 
			ParameterNumber:= MC_AxisParameter.AxisDec, 
			ReadMode:= 1 );
		fbAxisParamRead[4](
			Axis:= HardwareAxis, 
			Enable:=TRUE , 
			ParameterNumber:= MC_AxisParameter.AxisJerk, 
			ReadMode:= 1 );
		fbAxisParamRead[5](
			Axis:= HardwareAxis, 
			Enable:=TRUE , 
			ParameterNumber:= MC_AxisParameter.AxisMaxVelocity, 
			ReadMode:= 1 );
		fbAxisParamRead[6](
			Axis:= HardwareAxis, 
			Enable:=TRUE , 
			ParameterNumber:= MC_AxisParameter.AxisManualVelocityFast, 
			ReadMode:= 1 );
		fbAxisParamRead[7](
			Axis:= HardwareAxis, 
			Enable:=TRUE , 
			ParameterNumber:= MC_AxisParameter.AxisManualVelocitySlow, 
			ReadMode:= 1 );
		fbAxisParamRead[8](
			Axis:= HardwareAxis, 
			Enable:=TRUE , 
			ParameterNumber:= MC_AxisParameter.AxisEncoderModuloValue, 
			ReadMode:= 1 );			
		IF NOT (fbAxisParamRead[1].Busy AND fbAxisParamRead[1].Valid) AND NOT 
				(fbAxisParamRead[2].Busy AND fbAxisParamRead[2].Valid) AND NOT 
				(fbAxisParamRead[3].Busy AND fbAxisParamRead[3].Valid) AND NOT 
				(fbAxisParamRead[4].Busy AND fbAxisParamRead[4].Valid) AND NOT 
				(fbAxisParamRead[5].Busy AND fbAxisParamRead[5].Valid) AND NOT 
				(fbAxisParamRead[6].Busy AND fbAxisParamRead[6].Valid) AND NOT 
				(fbAxisParamRead[7].Busy AND fbAxisParamRead[7].Valid) AND NOT 
				(fbAxisParamRead[8].Busy AND fbAxisParamRead[8].Valid)	THEN
			nAxisCopy := 20;
		ELSIF fbAxisParamRead[1].Error OR fbAxisParamRead[2].Error OR fbAxisParamRead[3].Error OR fbAxisParamRead[4].Error OR fbAxisParamRead[5].Error OR fbAxisParamRead[6].Error OR fbAxisParamRead[7].Error OR fbAxisParamRead[8].Error THEN
			nAxisCopy := 40;
		END_IF
	20:	//write axis param
		fbWriteParam[1](
			Axis:=SimulationAxis , 
			Execute:= TRUE, 
			ParameterNumber:= MC_AxisParameter.AxisVeloMax, 
			Value:= fTestValue );
		fbWriteParam[2](
			Axis:=SimulationAxis , 
			Execute:= TRUE, 
			ParameterNumber:=  MC_AxisParameter.AxisAcc, 
			Value:=fbAxisParamRead[2].Value );
		fbWriteParam[3](
			Axis:=SimulationAxis , 
			Execute:= TRUE, 
			ParameterNumber:=  MC_AxisParameter.AxisDec, 
			Value:=fbAxisParamRead[3].Value );
		fbWriteParam[4](
			Axis:=SimulationAxis , 
			Execute:= TRUE, 
			ParameterNumber:= MC_AxisParameter.AxisJerk, 
			Value:=fbAxisParamRead[4].Value );
		fbWriteParam[5](
			Axis:=SimulationAxis , 
			Execute:= TRUE, 
			ParameterNumber:= MC_AxisParameter.AxisMaxVelocity, 
			Value:=fbAxisParamRead[5].Value );
		fbWriteParam[6](
			Axis:=SimulationAxis , 
			Execute:= TRUE, 
			ParameterNumber:= MC_AxisParameter.AxisManualVelocityFast, 
			Value:=fbAxisParamRead[6].Value );
		fbWriteParam[7](
			Axis:=SimulationAxis , 
			Execute:= TRUE, 
			ParameterNumber:= MC_AxisParameter.AxisManualVelocitySlow, 
			Value:=fbAxisParamRead[7].Value );
		fbWriteParam[8](
			Axis:=SimulationAxis , 
			Execute:= TRUE, 
			ParameterNumber:= MC_AxisParameter.AxisEncoderModuloValue, 
			Value:=fbAxisParamRead[8].Value );		
		IF 	fbWriteParam[1].Done AND fbWriteParam[2].Done AND fbWriteParam[3].Done AND fbWriteParam[4].Done AND fbWriteParam[5].Done AND fbWriteParam[6].Done AND fbWriteParam[7].Done AND fbWriteParam[8].Done THEN 
			bParamCopyComplete := TRUE;
			nAxisCopy := 25;
		ELSIF fbWriteParam[1].Error OR fbWriteParam[2].Error OR fbWriteParam[3].Error OR fbWriteParam[4].Error OR fbWriteParam[5].Error OR fbWriteParam[6].Error OR fbWriteParam[7].Error OR fbWriteParam[8].Error THEN
			nAxisCopy := 40;		
		END_IF
	25: // write the hardware axis position to the simulation axis		
		fbSetSimulationPosition(
								Axis:=SimulationAxis , 
								Execute:= TRUE, 
								Position:= HardwareAxis.NcToPlc.ActPos);
		IF fbSetSimulationPosition.Done THEN 
			nAxisCopy:= 30;
		ELSIF 	fbSetSimulationPosition.Error THEN
			nAxisCopy := 40;
		END_IF
	
	30: //set selected axis
		SelectedAxis REF= SimulationAxis;
		MotionControl();
	40: //reset FB's execute and retry
		nAxisCopy :=0;
END_CASE

//SelectedAxis REF= SimulationAxis;
//MotionControl();
END_METHOD

METHOD StandardOperation : BOOL
VAR_INPUT
END_VAR
SelectedAxis REF= HardwareAxis;
nAxisCopy :=0;
MotionControl();
END_METHOD

METHOD Stop : BOOL
fbAxisHalt.Execute := TRUE;
END_METHOD

PROPERTY Stopped : BOOL
GET
Stopped := bStopped;//Axis1.Status.StandStill;
END_GET
END_PROPERTY

PROPERTY TargetVelocity : LREAL
GET
TargetVelocity : fTargetVelocity;
END_GET
SET
fTargetVelocity : TargetVelocity;
END_SET
END_PROPERTY

METHOD Uninhibit : BOOL
VAR_INPUT
END_VAR
fOverride := 100;
END_METHOD

END_FUNCTION_BLOCK

// ---- Base/03_Utilities/03_HMI_Connections/FB_MainHMI_Connection.TcPOU
FUNCTION_BLOCK FB_MainHMI_Connection
VAR_IN_OUT
END_VAR
VAR_INPUT
	sTopLevelMachine : STRING;
END_VAR
VAR_OUTPUT
END_VAR
VAR
	fbModuleTree : FB_Tree_IndexBased;
	a_stMachineTreeNodes	: ARRAY[0..63] OF ST_Tree_IndexBased_Node;
	bInitialized : BOOL;

END_VAR

IF NOT bInitialized THEN
	(*
	sTopLevelMachine := 'My machine';		//TODO: Proper implementation of auto-generating tree structure
	fbModuleTree(a_stNodes := stMachineTreeNodes, sHead := sTopLevelMachine);
	fbModuleTree.AddNodeAsChildByName(sNewName := 'EM1', sParentName := 'My machine');
	fbModuleTree.AddNodeAsChildByName(sNewName := 'CM1', sParentName := 'EM1');
	fbModuleTree.AddNodeAsChildByName(sNewName := 'CP1', sParentName := 'CM1');
	fbModuleTree.AddNodeAsChildByName(sNewName := 'CP2', sParentName := 'CM1');
	fbModuleTree.AddNodeAsChildByName(sNewName := 'CM2', sParentName := 'EM1');
	fbModuleTree.AddNodeAsChildByName(sNewName := 'CM3', sParentName := 'EM1');
	fbModuleTree.AddNodeAsChildByName(sNewName := 'CP3', sParentName := 'CM3');
	fbModuleTree.AddNodeAsChildByName(sNewName := 'EM2', sParentName := 'My machine');
	fbModuleTree.AddNodeAsChildByName(sNewName := 'CM4', sParentName := 'EM2');
	fbModuleTree.AddNodeAsChildByName(sNewName := 'CM5', sParentName := 'EM2');
	fbModuleTree.AddNodeAsChildByName(sNewName := 'CP4', sParentName := 'CM5');
	fbModuleTree.AddNodeAsChildByName(sNewName := 'CP5', sParentName := 'CM5');
	fbModuleTree.AddNodeAsChildByName(sNewName := 'CP10', sParentName := 'CM5');
	fbModuleTree.AddNodeAsChildByName(sNewName := 'CP11', sParentName := 'CM5');
	fbModuleTree.AddNodeAsChildByName(sNewName := 'CP12', sParentName := 'CM5');
	fbModuleTree.AddNodeAsChildByName(sNewName := 'CM6', sParentName := 'EM2');
	fbModuleTree.AddNodeAsChildByName(sNewName := 'CM7', sParentName := 'EM2');
	fbModuleTree.AddNodeAsChildByName(sNewName := 'CP7', sParentName := 'CM7');
	fbModuleTree.AddNodeAsChildByName(sNewName := 'EM3', sParentName := 'My machine');
	fbModuleTree.AddNodeAsChildByName(sNewName := 'CM8', sParentName := 'EM3');
	fbModuleTree.AddNodeAsChildByName(sNewName := 'CM9', sParentName := 'EM3');
	fbModuleTree.AddNodeAsChildByName(sNewName := 'CP8', sParentName := 'CM9');
	fbModuleTree.AddNodeAsChildByName(sNewName := 'CP9', sParentName := 'CM9');
	fbModuleTree.AddNodeAsChildByName(sNewName := 'EM4', sParentName := 'My machine');
	*)
	fbModuleTree(a_stNodes := a_stMachineTreeNodes, sHead := sTopLevelMachine);
	
	bInitialized := TRUE;
END_IF

PROPERTY DataStructure_Adder : ITF_Tree_IndexBased
GET
DataStructure_Adder := fbModuleTree;
END_GET
END_PROPERTY

END_FUNCTION_BLOCK

// ---- Base/03_Utilities/02_DataStructures/01_Tree/01_Tree_IndexBased/FB_Tree_IndexBased.TcPOU
FUNCTION_BLOCK FB_Tree_IndexBased IMPLEMENTS ITF_Tree_IndexBased
VAR_IN_OUT
	a_stNodes : ARRAY[0..63] OF ST_Tree_IndexBased_Node;
END_VAR
VAR_INPUT
	sHead : STRING;
END_VAR
VAR
	bInitialized 	: BOOL;
	nNodeCount 		: DINT;
	nNewNodeIndex	: DINT;
	nHeadIndex		: DINT;
	
	//"Temp" variables for use in AddNodeAsChildByName
	nParentIndex 	: DINT;
	nChildCount		: DINT;
END_VAR

IF NOT bInitialized THEN
	initialize();
END_IF

METHOD AddNodeAsChildByName : BOOL
VAR_INPUT
	sNewName 	: STRING;
	sParentName	: STRING;
END_VAR
nParentIndex := GetIndexByName(sParentName);		//Find the index value of the designated parent node
nChildCount := a_stNodes[nParentIndex].nChildCount;
IF nParentIndex >= 0 THEN	//If GetIndex was successful
	IF (a_stNodes[nParentIndex].nChildCount < 64) THEN	//TODO: Proper Constant bound definition	//If the parent is not at max child count
		a_stNodes[nNewNodeIndex].sName := sNewName;		//assign new node name to next empty node in list
		a_stNodes[nNewNodeIndex].nParent := nParentIndex;	//assign the parent node to the new child node
		a_stNodes[nNewNodeIndex].nDepth := a_stNodes[nParentIndex].nDepth + 1;
		a_stNodes[nParentIndex].a_nChildren[nChildCount] := nNewNodeIndex;		//assign the new node location as the next child in the parent
		nNewNodeIndex := nNewNodeIndex + 1;		//Increment to next empty node
		a_stNodes[nParentIndex].nChildCount := nChildCount + 1;
	END_IF
END_IF
END_METHOD

METHOD GetIndexByName : DINT
VAR_INPUT
	sName : STRING;
END_VAR
VAR
	i : DINT;
END_VAR
FOR i := 0 TO nNodeCount DO
	IF a_stNodes[i].sName = sName THEN
		GetIndexByName := i;
		RETURN;
	END_IF
END_FOR

GetIndexByName := -1;
END_METHOD

METHOD PRIVATE initialize : BOOL
VAR_INPUT
END_VAR
//nNodeCount := UPPER_BOUND(a_stNodes,1) - LOWER_BOUND(a_stNodes,1) + 1;
nNodeCount := 64;
IF nNodeCount >= 0 THEN
	nHeadIndex := 0;//LOWER_BOUND(a_stNodes,1);
	a_stNodes[nHeadIndex].sName := sHead;
	a_stNodes[nHeadIndex].nDepth := 0;
	a_stNodes[nHeadIndex].nParent := -1;
	nNewNodeIndex := nHeadIndex + 1;
END_IF
END_METHOD

END_FUNCTION_BLOCK

// ---- Base/01_PML/01_Module/04_SequenceControl/F_CommandAllSequences.TcPOU
FUNCTION F_CommandAllSequences : BOOL
VAR_IN_OUT
	itfSequenceArray	: ARRAY[*] OF ITF_ModuleSequenceControl;
END_VAR
VAR_INPUT
	eCommand			: E_ModuleSequenceCommand;
	nSubCount			: UDINT;
END_VAR
VAR
	i:	UDINT;
END_VAR

CASE eCommand OF
	E_ModuleSequenceCommand.Clear:
		FOR i := 1 TO nSubCount DO
			itfSequenceArray[i].ClearSequence();
		END_FOR
		
	E_ModuleSequenceCommand.Disable:
		FOR i := 1 TO nSubCount DO
			itfSequenceArray[i].DisableSequence();
		END_FOR
	
	E_ModuleSequenceCommand.Enable:
		FOR i := 1 TO nSubCount DO
			itfSequenceArray[i].EnableSequence();
		END_FOR
	
	E_ModuleSequenceCommand.Reset:
		FOR i := 1 TO nSubCount DO
			itfSequenceArray[i].ResetSequence();
		END_FOR
	
	E_ModuleSequenceCommand.Resume:
		FOR i := 1 TO nSubCount DO
			itfSequenceArray[i].ResumeSequence();
		END_FOR
	
	E_ModuleSequenceCommand.Start:
		FOR i := 1 TO nSubCount DO
			itfSequenceArray[i].StartSequence();
		END_FOR
	
END_CASE

END_FUNCTION

// ---- Base/01_PML/99_Templates/01_ModuleTemplate/FB_ApplicationModule_TEMPLATE.TcPOU
(*
	Use this module to copy to Application and use for a machine
	
	Remove the ABSTRACT from the definition and refactor(Rename) the FB
*)

FUNCTION_BLOCK ABSTRACT FB_ApplicationModule_TEMPLATE EXTENDS FB_PMLModuleBase
VAR
	//Define the Sub modules here for this module.  Also set the Interfaces in the initialize method.
	//fbSubModule1				: FB_ApplicationModule_TEMPLATE;		// Sub module instantiation
	//fbSubModule2				: FB_ApplicationModule_TEMPLATE;		// Sub module instantiation
	
	//temporary array of module base interfaces to be copied over to the base class a_itfPackMLBase variable
	a_itfPackMLBase_init		: ARRAY[1..MAX_NO_OF_SUBUNITS] OF ITF_PMLModuleBase (*:= [fbSubModule1, fbSubModule2,*);

	// Other machine specific variables here
END_VAR

//*********************************************************
// Code implementation only in Execute() method for consistency with templates
//*********************************************************

// 
// Cyclic Code
METHOD CyclicLogic
VAR
	i								: UDINT;		//Generic iteration value
END_VAR
// Main loop of the parent module
SUPER^.CyclicLogic();
END_METHOD

METHOD Initialize
VAR
	i								: UDINT;		//Generic iteration value
END_VAR

// Define the interfaces to the different subunits (Must take place before SUPER^.initialize call)
FOR i := 1 TO MAX_NO_OF_SUBUNITS DO
	a_itfPackMLBase[i] := a_itfPackMLBase_init[i];
END_FOR


// Init of the parent class object (Must be called AFTER most local init code, since the sub module interface array assignments should be made here, and then operated on within the module base init
SUPER^.Initialize();
END_METHOD

END_FUNCTION_BLOCK

// ---- Base/02_Components/02_Axes/02_Homing/FB_Axis_HomeToSensor.TcPOU
FUNCTION_BLOCK FB_Axis_HomeToSensor EXTENDS FB_AxisBase
VAR_INPUT
END_VAR
VAR_OUTPUT
END_VAR
VAR
	//I/O definitions
	fbHomeSensor		: FB_Sensor;
	
	//Internal Property Variables
	fHomePositionSetpoint		: LREAL := 0;
	bHomeSensorStatus			: BOOL;
END_VAR

METHOD Home : BOOL
VAR_INPUT
END_VAR
SUPER^.Home();

IF NOT bActive THEN
	fbAxisHome.Execute := TRUE;
END_IF
END_METHOD

PROPERTY HomePositionSetpoint : LREAL
GET
HomePositionSetpoint := fHomePositionSetpoint;
END_GET
SET
fHomePositionSetpoint := HomePositionSetpoint;
END_SET
END_PROPERTY

PROPERTY HomeSensorStatus : BOOL
GET
HomeSensorStatus := bHomeSensorStatus;
END_GET
END_PROPERTY

METHOD Monitoring : BOOL
SUPER^.Monitoring();

bHomeSensorStatus := fbHomeSensor.Active;
END_METHOD

METHOD MotionControl : BOOL
VAR_INPUT
END_VAR
SUPER^.MotionControl();

//Performs a simple home-to sensor sequence when commanded by a "Home" Method call
fbAxisHome(
	Axis:= SelectedAxis,
	Position:= fHomePositionSetpoint, 
	HomingMode:= MC_HomingMode.MC_DefaultHoming, 
	BufferMode:= MC_BufferMode.MC_Aborting,
	bCalibrationCam := bHomeSensorStatus);

fbAxisHome.Execute := FALSE;
END_METHOD

END_FUNCTION_BLOCK

// ---- Base/02_Components/02_Axes/03_MotionType/FB_Axis_Continuous_HomeToSensor.TcPOU
FUNCTION_BLOCK FB_Axis_Continuous_HomeToSensor EXTENDS FB_Axis_HomeToSensor IMPLEMENTS ITF_Axis_Continuous
VAR_INPUT
END_VAR
VAR_OUTPUT
END_VAR
VAR
	//Internal Property Variables
	fModuloPosition		: LREAL;
	fModuloFactor		: LREAL;
END_VAR

PROPERTY ModuloFactor : LREAL
GET
ModuloFactor := fModuloFactor;
END_GET
END_PROPERTY

PROPERTY ModuloPosition : LREAL
GET
ModuloPosition := fModuloPosition;
END_GET
END_PROPERTY

METHOD Monitoring : BOOL
SUPER^.Monitoring();

fModuloPosition := SelectedAxis.NcToPlc.ModuloActPos;

IF fbWriteParameter.Done AND fbWriteParameter.ParameterNumber = MC_AxisParameter.AxisEncoderModuloValue THEN
	fModuloFactor := fbWriteParameter.Value;
END_IF

IF fbWriteParameter.Error AND NOT fbAxisBaseAlarms[E_AxisBase.WriteParameterError].bRaised THEN
	bError := TRUE;
	nErrorID := E_AxisBase.WriteParameterError;
	sTemp := UDINT_TO_STRING(fbWriteParameter.ErrorID);
	fbAxisBaseAlarms[E_AxisBase.WriteParameterError].ipArguments.Clear().AddString(sName).AddString(sTemp);
	fbAxisBaseAlarms[E_AxisBase.WriteParameterError].Raise(0);
ELSIF NOT fbAxisPower.Error AND fbAxisBaseAlarms[E_AxisBase.WriteParameterError].bRaised THEN
	fbAxisBaseAlarms[E_AxisBase.WriteParameterError].Clear(0,0);
END_IF
END_METHOD

METHOD SetAxisModuloFactor : BOOL
VAR_INPUT
	fSetAxisModuloFactor		: LREAL;
END_VAR
IF NOT bActive THEN
	IF NOT fbWriteParameter.Busy THEN
	fbWriteParameter(
						Axis:= SelectedAxis, 
						Execute:= TRUE, 
						ParameterNumber:= MC_AxisParameter.AxisEncoderModuloValue, 
						Value:= fSetAxisModuloFactor, 
						Done=> , 
						Busy=> , 
						Error=> , 
						ErrorID=> );
	END_IF
ELSE
	//TODO: Messaging for "Axis not ready for parameter write"
END_IF
END_METHOD

END_FUNCTION_BLOCK

// ---- Base/02_Components/02_Axes/03_MotionType/FB_Axis_Discrete_HomeToSensor.TcPOU
FUNCTION_BLOCK FB_Axis_Discrete_HomeToSensor EXTENDS FB_Axis_HomeToSensor
VAR_INPUT
END_VAR
VAR_OUTPUT
END_VAR
VAR
	//If preferred, initialize upper limit to a value less than the lower limit to prevent operation until proper soft limits have been configured
	fLowerTravelLimit			: LREAL := -1.7976931348623158E+308; //(Minimum LREAL value)
	fUpperTravelLimit			: LREAL := 1.7976931348623158E+308;	//(Maximum LREAL value)
	fPosition_1					: LREAL;
	fPosition_2					: LREAL;
	fPosition_3					: LREAL;
	
END_VAR

METHOD Home : BOOL
VAR_INPUT
END_VAR
SUPER^.Home();

IF NOT bActive THEN
	fbAxisHome.Execute := TRUE;
END_IF
END_METHOD

PROPERTY LowerTravelLimit : LREAL
GET
LowerTravelLimit := fLowerTravelLimit;
END_GET
SET
fLowerTravelLimit := LowerTravelLimit;
END_SET
END_PROPERTY

METHOD Monitoring : BOOL
VAR_INPUT
END_VAR
SUPER^.Monitoring();

//Monitor soft travel limits
IF fPosition >= fUpperTravelLimit AND fPositionSetpoint > fUpperTravelLimit THEN
	Inhibit();
	//TODO: log specific message for soft limit reached
END_IF

IF fPosition <= fLowerTravelLimit AND fPositionSetpoint < fLowerTravelLimit THEN
	Inhibit();
	//TODO: log specific message for soft limit reached
END_IF

IF  fOverride = 0 AND fPositionSetpoint < fUpperTravelLimit AND fPositionSetpoint > fLowerTravelLimit THEN
	Uninhibit();
	//TODO: log specific message for soft limit reached
END_IF
END_METHOD

METHOD MotionControl : BOOL
VAR_INPUT
END_VAR
SUPER^.MotionControl();

//Performs a simple home-to sensor sequence when commanded by a "Home" Method call
fbAxisHome(
	Axis:= SelectedAxis,
	Position:= fHomePositionSetpoint, 
	HomingMode:= MC_HomingMode.MC_DefaultHoming, 
	BufferMode:= MC_BufferMode.MC_Aborting,
	bCalibrationCam := bHomeSensorStatus);

fbAxisHome.Execute := FALSE;
END_METHOD

PROPERTY Position_1 : LREAL
GET
Position_1 := fPosition_1;
END_GET
SET
fPosition_1 := Position_1;
END_SET
END_PROPERTY

PROPERTY Position_2 : LREAL
GET
Position_2 := fPosition_2;
END_GET
SET
fPosition_2 := Position_2;
END_SET
END_PROPERTY

PROPERTY Position_3 : LREAL
GET
Position_3 := fPosition_3;
END_GET
SET
fPosition_3 := Position_3;
END_SET
END_PROPERTY

PROPERTY UpperTravelLimit : LREAL
GET
UpperTravelLimit := fUpperTravelLimit;
END_GET
SET
fUpperTravelLimit := UpperTravelLimit;
END_SET
END_PROPERTY

END_FUNCTION_BLOCK

// ---- Application/01_Application_Level_Items/99_VISU/V_Application.TcVIS
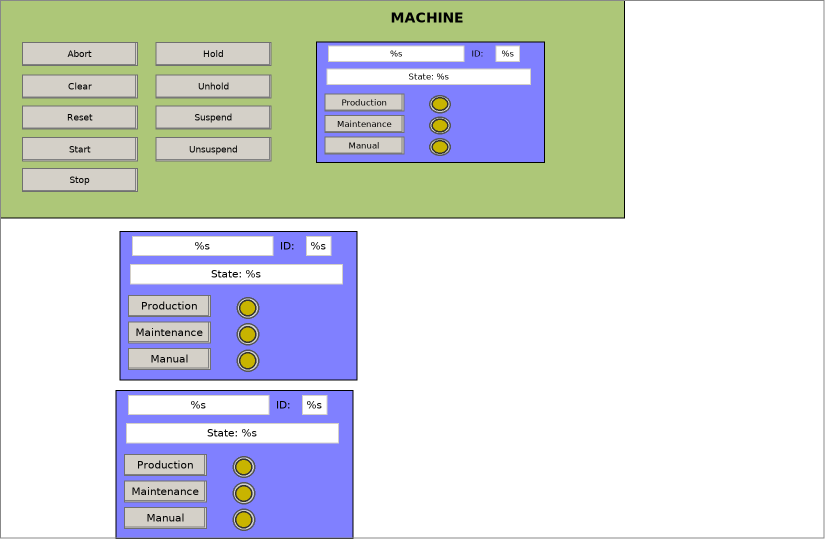
VISUALIZATION V_Application  // 825x539
    Frame (0,0 825x218)
        shows V_MachineModule(stVisu := MAIN.fbMyMachine.stPMLModuleBaseVISU)
    Frame (110,222 247x158)
        shows V_Module(stVisu := MAIN.fbMyMachine.fbEquipmentModule1.stPMLModuleBaseVISU)
    Frame (106,381 247x158)
        shows V_Module(stVisu := MAIN.fbMyMachine.fbEquipmentModule1.fb_EM1_ControlModule1.stPMLModuleBaseVISU)
END_VISUALIZATION

// ---- Base/01_PML/01_Module/05_Visualizations/V_Module.TcVIS
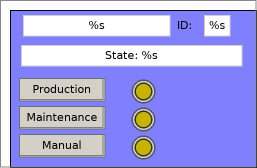
VISUALIZATION V_Module  // 257x168
VAR_IN_OUT
	stVisu				: ST_PMLModuleBaseVISU;
END_VAR
    RoundedRectangle (10,10 247x158)
    Textfield (23,15 147x21), "%s", text variable: stVisu.sModuleName
    Textfield (204,15 26x21), "%s", text variable: stVisu.nModuleID
    Label (165,14 39x23), "ID:"
    Textfield (21,45 221x21), "State: %s", text variable: stVisu.eState
    Button (19,78 86x23), "Production"
        tap stVisu.bProductionPressed
    Button (19,106 86x23), "Maintenance"
        tap stVisu.bMaintenancePressed
    Button (19,134 86x23), "Manual"
        tap stVisu.bManualPressed
    Lamp1 (130,78 27x27), variable: stVisu.eMode = E_PMLProtectedUnitMode.ePMLProtUnitMode_Production, style: Lamp-Lamp1-Yellow
    Lamp1 (130,106 27x27), variable: stVisu.eMode = E_PMLProtectedUnitMode.ePMLProtUnitMode_Maintenance, style: Lamp-Lamp1-Yellow
    Lamp1 (130,134 27x27), variable: stVisu.eMode = E_PMLProtectedUnitMode.ePMLProtUnitMode_Manual, style: Lamp-Lamp1-Yellow
END_VISUALIZATION

// ---- Base/01_PML/03_Visualizations/V_MachineModule.TcVIS
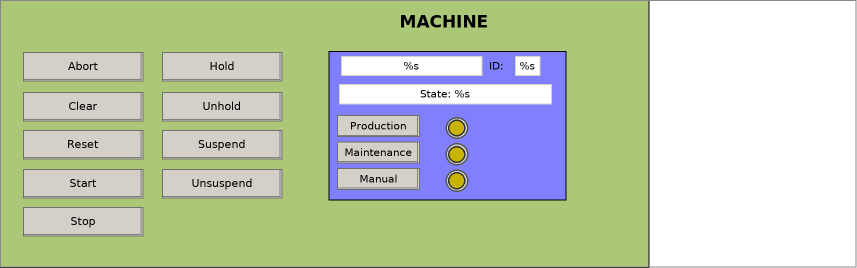
VISUALIZATION V_MachineModule  // 857x268
VAR_IN_OUT
	stVisu				: ST_PMLModuleBaseVISU;
END_VAR
    RoundedRectangle (0,0 649x268)
    Button (23,52 120x29), "Abort"
        tap stVisu.bAbortPressed
    Button (23,92 120x29), "Clear"
        tap stVisu.bClearPressed
    Button (23,130 120x29), "Reset"
        tap stVisu.bResetPressed
    Button (23,169 120x29), "Start"
        tap stVisu.bStartPressed
    Button (23,207 120x29), "Stop"
        tap stVisu.bStopPressed
    Button (162,52 120x29), "Hold"
        tap stVisu.bHoldPressed
    Button (162,92 120x29), "Unhold"
        tap stVisu.bUnholdPressed
    Button (162,130 120x29), "Suspend"
        tap stVisu.bSuspendPressed
    Button (162,169 120x29), "Unsuspend"
        tap stVisu.bUnsuspendPressed
    Frame (319,42 247x158)
        shows V_Module(stVisu := stVisu)
    Label (31,3 826x37), "MACHINE"
END_VISUALIZATION

// ---- GlobalTextList.TcGTLO
TEXTLIST GlobalTextList
  685 = '%s'
  680 = 'Abort'
  407 = 'Active'
  255 = 'ActiveAlarm'
  756 = 'AirOK'
  781 = 'Alarm'
  452 = 'Clear'
  136 = 'eState'
  744 = 'Hold'
  789 = 'ID'
  194 = 'ID:'
  12 = 'itfPMLBase.'
  347 = 'MACHINE'
  568 = 'Machine Name: %s'
  46 = 'Maintenance'
  904 = 'Manual'
  667 = 'Mode: %s'
  962 = 'Name'
  613 = 'PowerOK'
  929 = 'Production'
  181 = 'Reset'
  77 = 'Start'
  516 = 'State: %s'
  828 = 'Stop'
  806 = 'Suspend'
  197 = 'Unhold'
  515 = 'UnitModeCurrent'
  832 = 'Unsuspend'
END_TEXTLIST
